FUNCTION ARR08X_TO_BYTE
  (* Standard: 61499-1; Description: Copyright (c) 2024 HR Agrartechnik GmbH This program and the accompanying materials are made available under the terms of the Eclipse Public License 2.0 which is available at https://www.eclipse.org/legal/epl-2.0/ SPDX-License-Identifier: EPL-2.0 *)
  (* Version 1.0, 2024-02-22, Franz Höpfinger, HR Agrartechnik GmbH *)
  PACKAGE logiBUS::utils::conversion::arr::assembling;
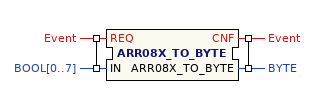
  EVENT_INPUT
    REQ WITH IN;
  END_EVENT
  EVENT_OUTPUT
    CNF WITH ARR08X_TO_BYTE;
  END_EVENT
  VAR_INPUT
    IN : ARRAY [0..7] OF BOOL; (* ARR08B Input *)
  END_VAR
  VAR_OUTPUT
    ARR08X_TO_BYTE : BYTE;
  END_VAR
  BODY IN ST:
PACKAGE logiBUS::utils::conversion::arr::assembling;

FUNCTION ARR08X_TO_BYTE : BYTE

VAR_INPUT
	IN : ARRAY[0..7] OF BOOL; // ARR08B Input
END_VAR

(* this Function extracts the 8 Bits from a byte *)
ARR08X_TO_BYTE.0 := IN[0];
ARR08X_TO_BYTE.1 := IN[1];
ARR08X_TO_BYTE.2 := IN[2];
ARR08X_TO_BYTE.3 := IN[3];
ARR08X_TO_BYTE.4 := IN[4];
ARR08X_TO_BYTE.5 := IN[5];
ARR08X_TO_BYTE.6 := IN[6];
ARR08X_TO_BYTE.7 := IN[7];

END_FUNCTION
  END_BODY
END_FUNCTION
